// TIA Portal V20 export
FUNCTION_BLOCK "LER_visionHistory"   // FB80, LAD
// stored: Access Published, MemoryReserve 100, SetENOAutomatically false
   VAR_INPUT
      save : Bool;
      result { ExternalAccessible := 'False'; ExternalVisible := 'False'; ExternalWritable := 'False'} : "LER_typePartData";
   END_VAR
   VAR_IN_OUT
      dataHistory : "LER_typeVisionHistory";
   END_VAR
   VAR
      statDeleteData : "LER_typeVisionHistory";
      statTonTimer { S7_SetPoint := 'True'} : Array[0..9] of TON_TIME;
      statTrigger : Array[0..9] of Bool;
      statComplete : Bool;
   END_VAR
   VAR_TEMP
      tempRetVal : Array[0..9] of Int;
   END_VAR
   VAR_TEMP   // added for the SCL form of the ladder/FBD networks
      _w1 : Bool;
   END_VAR
BEGIN

REGION Network 1: History
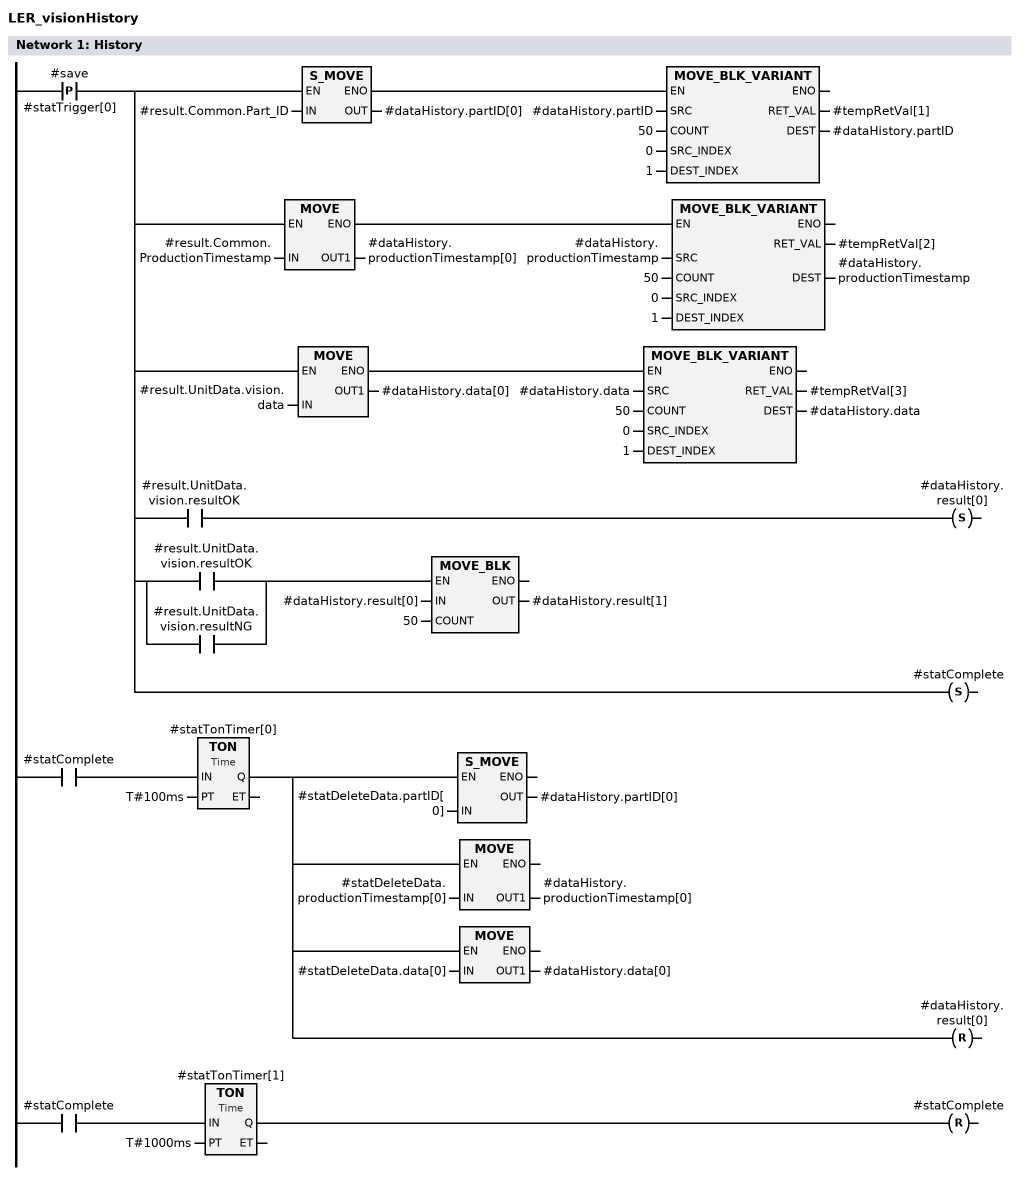
   #_w1 := #save AND NOT #statTrigger[0];   // rising edge of #save
   #statTrigger[0] := #save;
   IF #_w1 THEN
       #dataHistory.partID[0] := #result.Common.Part_ID;
       #tempRetVal[1] := MOVE_BLK_VARIANT(SRC := #dataHistory.partID,
                               COUNT := 50,
                               SRC_INDEX := 0,
                               DEST_INDEX := 1,
                               DEST => #dataHistory.partID);
       #dataHistory.productionTimestamp[0] := #result.Common.ProductionTimestamp;
       #tempRetVal[2] := MOVE_BLK_VARIANT(SRC := #dataHistory.productionTimestamp,
                               COUNT := 50,
                               SRC_INDEX := 0,
                               DEST_INDEX := 1,
                               DEST => #dataHistory.productionTimestamp);
       #dataHistory.data[0] := #result.UnitData.vision.data;
       #tempRetVal[3] := MOVE_BLK_VARIANT(SRC := #dataHistory.data,
                               COUNT := 50,
                               SRC_INDEX := 0,
                               DEST_INDEX := 1,
                               DEST => #dataHistory.data);
   END_IF;
   IF #_w1 AND #result.UnitData.vision.resultOK THEN #dataHistory.result[0] := TRUE; END_IF;
   IF #_w1 AND (#result.UnitData.vision.resultOK OR #result.UnitData.vision.resultNG) THEN
       MOVE_BLK(IN := #dataHistory.result[0], COUNT := 50, OUT => #dataHistory.result[1]);
   END_IF;
   IF #_w1 THEN #statComplete := TRUE; END_IF;
   #statTonTimer[0].TON(IN := #statComplete, PT := T#100ms);
   IF #statTonTimer[0].Q THEN
       #dataHistory.partID[0] := #statDeleteData.partID[0];
       #dataHistory.productionTimestamp[0] := #statDeleteData.productionTimestamp[0];
       #dataHistory.data[0] := #statDeleteData.data[0];
       #dataHistory.result[0] := FALSE;
   END_IF;
   #statTonTimer[1].TON(IN := #statComplete, PT := T#1000ms);
   IF #statTonTimer[1].Q THEN #statComplete := FALSE; END_IF;
END_REGION
END_FUNCTION_BLOCK
